// TIA Portal V17 export
// export: Created 2025-05-08T13:17:41.9955383Z, ExportSetting WithDefaults, DisplayName Totally Integrated Automation Portal, DisplayVersion V17 Update 8, DisplayName TIA Portal Openness, DisplayVersion V17 Update 8, DisplayName TIA Portal Version Control Interface, DisplayVersion V17, DisplayName SINAMICS Startdrive Advanced, DisplayVersion V17 SP2, DisplayName SINAMICS Startdrive G110M, G120, G120C, G120D, G120P, G115D, DisplayVersion V17 SP2, DisplayName SINAMICS Startdrive G130, G150, S120, S150, SINAMICS MV, S210, DisplayVersion V17 SP2, DisplayName STEP 7 Professional, DisplayVersion V17 Update 8, DisplayName SINUMERIK ONE STEP 7 Toolbox, DisplayVersion V17 Update 12, DisplayName SINUMERIK 840D sl STEP 7 Toolbox, DisplayVersion V17 Update 12, DisplayName STEP 7 Safety, DisplayVersion V17 Update 6, DisplayName WinCC Advanced, DisplayVersion V17 Update 8
FUNCTION "FC2001_AUTO_SINGLE_SEMI_MANUAL" : Void   // FC2001, LAD
{ S7_Optimized_Access := 'FALSE' }
AUTHOR : ETXETAR
VERSION : 1.0
// stored: AutoNumber false, IsIECCheckEnabled false, SetENOAutomatically false, UDAEnableTagReadback false
   VAR_TEMP
      O_BYTE_0 : Struct   // OPTIONS BYTE 0
         CHANGE_MODE_SEOC_ALARM : Bool;   // CHANGE MODE SEOC ALARM OPTION
         MODE_SELECTED_MEMORY : Bool;   // MODE SELECTED MEMORY OPTION
      END_STRUCT;
      MG1_INPUTS : Struct
         MANUAL : Bool;   // MANUAL INPUT
         SEMIAUTO : Bool;   // SEMIAUTO INPUT
         AUTOMATIC : Bool;   // AUTOMATIC INPUT
         SINGLE : Bool;   // SINGLE INPUT
         NO_MODE : Bool;   // NO MODE INPUT
         JOG : Bool;   // JOG INPUT
         "TOOL CHANGE" : Bool;   // TOOL CHANGE INPUT
      END_STRUCT;
      MG2_INPUTS : Struct
         MANUAL : Bool;   // MANUAL INPUT
         SEMIAUTO : Bool;   // SEMIAUTO INPUT
         AUTOMATIC : Bool;   // AUTOMATIC INPUT
         SINGLE : Bool;   // SINGLE INPUT
         NO_MODE : Bool;   // NO MODE INPUT
         JOG : Bool;   // JOG INPUT
         "TOOL CHANGE" : Bool;   // TOOL CHANGE INPUT
      END_STRUCT;
   END_VAR
   VAR CONSTANT
      FC_NUMBER : Int := 2001;   // NUMBER
   END_VAR
BEGIN

REGION Network 1: OPTIONS OFF
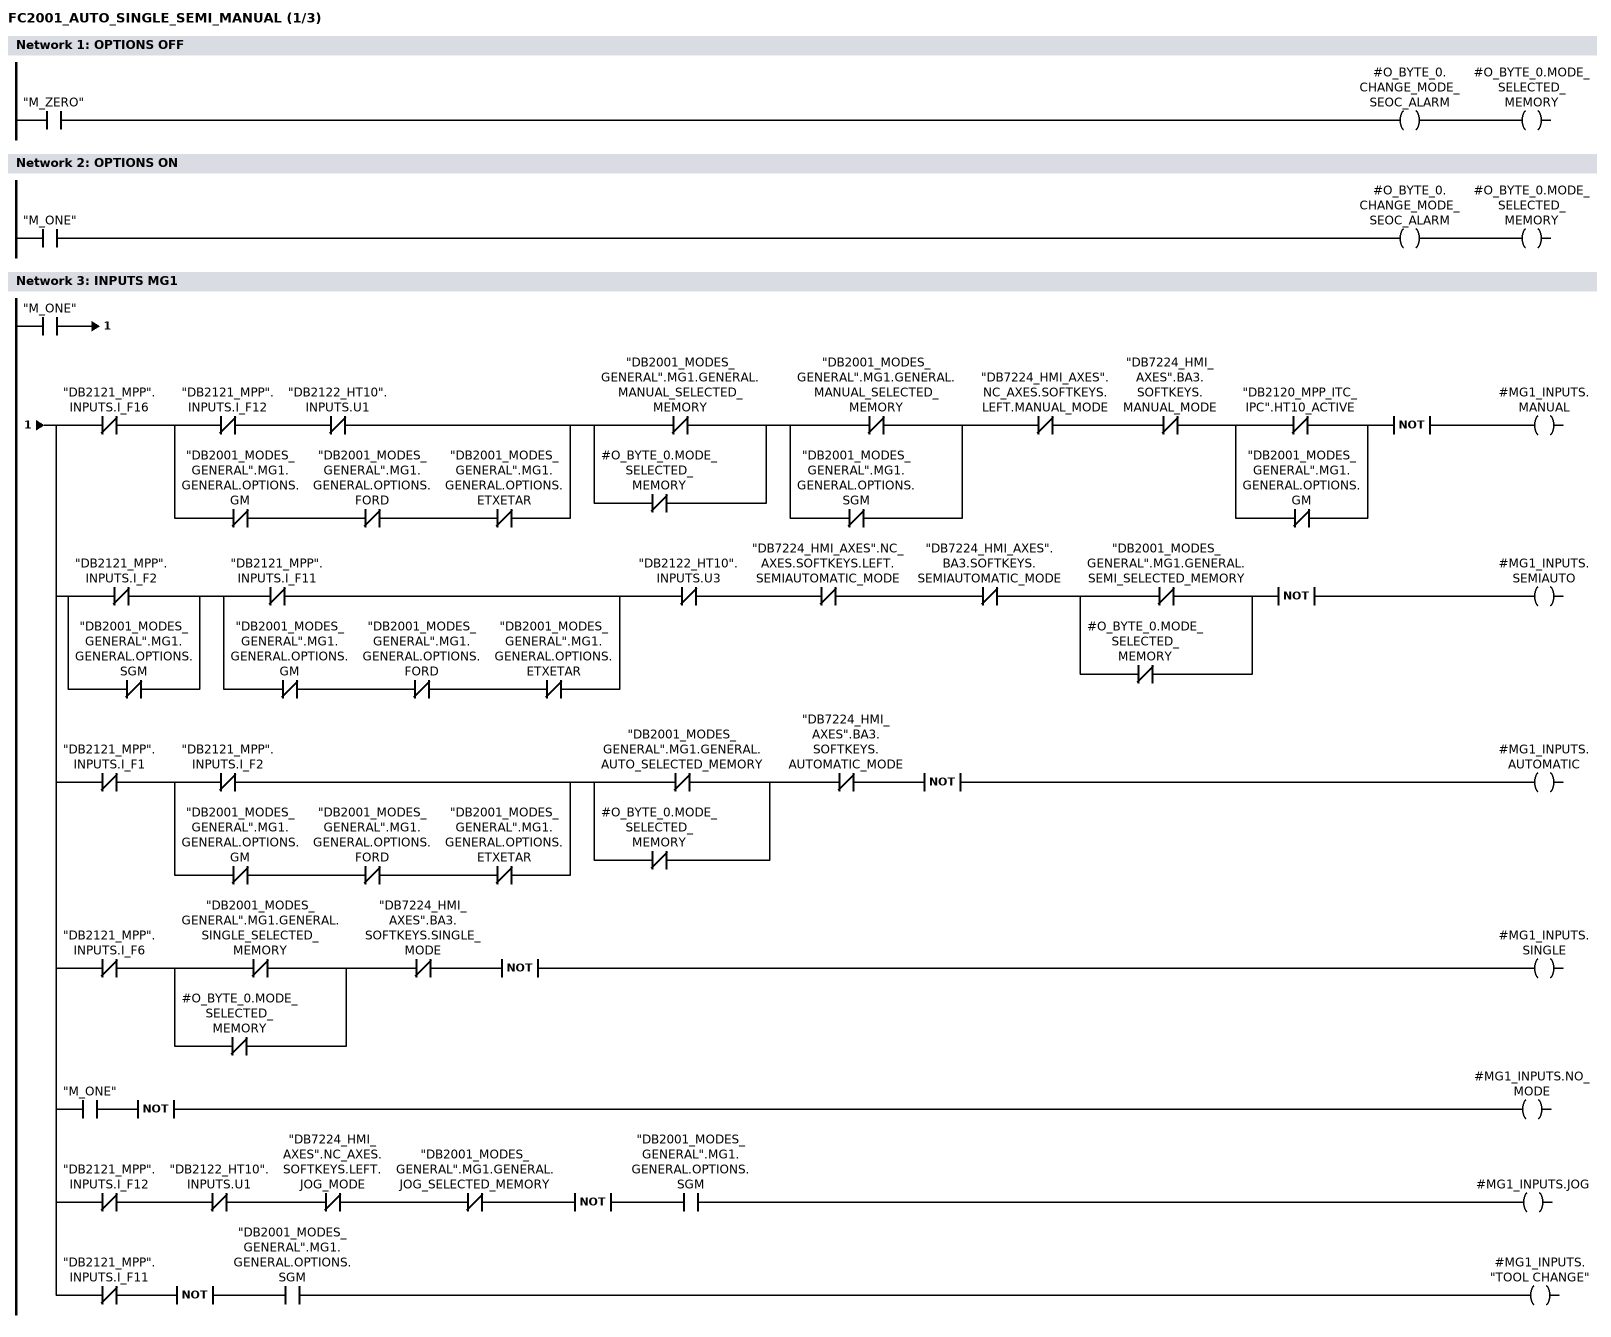
   RUNG wire#powerrail
      Contact( "M_ZERO" )
      Coil( #O_BYTE_0.CHANGE_MODE_SEOC_ALARM )
      Coil( #O_BYTE_0.MODE_SELECTED_MEMORY )
   END_RUNG
   // the same network as SCL:
   #O_BYTE_0.CHANGE_MODE_SEOC_ALARM := "M_ZERO";
   #O_BYTE_0.MODE_SELECTED_MEMORY := "M_ZERO";
END_REGION

REGION Network 2: OPTIONS ON
   RUNG wire#powerrail
      Contact( "M_ONE" )
      Coil( #O_BYTE_0.CHANGE_MODE_SEOC_ALARM )
      Coil( #O_BYTE_0.MODE_SELECTED_MEMORY )
   END_RUNG
   // the same network as SCL:
   #O_BYTE_0.CHANGE_MODE_SEOC_ALARM := "M_ONE";
   #O_BYTE_0.MODE_SELECTED_MEMORY := "M_ONE";
END_REGION

REGION Network 3: INPUTS MG1
   RUNG wire#powerrail
      Contact( "M_ONE" )
      wire#w1
      I_Contact( "DB2121_MPP".INPUTS.I_F16 )
      wire#w2
      I_Contact( "DB2121_MPP".INPUTS.I_F12 )
      I_Contact( "DB2122_HT10".INPUTS.U1 )
      wire#w3
      I_Contact( "DB2001_MODES_GENERAL".MG1.GENERAL.MANUAL_SELECTED_MEMORY )
      wire#w4
      I_Contact( "DB2001_MODES_GENERAL".MG1.GENERAL.MANUAL_SELECTED_MEMORY )
      wire#w5
      I_Contact( "DB7224_HMI_AXES".NC_AXES.SOFTKEYS.LEFT.MANUAL_MODE )
      I_Contact( "DB7224_HMI_AXES".BA3.SOFTKEYS.MANUAL_MODE )
      wire#w6
      I_Contact( "DB2120_MPP_ITC_IPC".HT10_ACTIVE )
      wire#w7
      Not()
      Coil( #MG1_INPUTS.MANUAL )
   END_RUNG
   RUNG wire#w2
      I_Contact( "DB2001_MODES_GENERAL".MG1.GENERAL.OPTIONS.GM )
      I_Contact( "DB2001_MODES_GENERAL".MG1.GENERAL.OPTIONS.FORD )
      I_Contact( "DB2001_MODES_GENERAL".MG1.GENERAL.OPTIONS.ETXETAR )
   END_RUNG wire#w3
   RUNG wire#w3
      I_Contact( #O_BYTE_0.MODE_SELECTED_MEMORY )
   END_RUNG wire#w4
   RUNG wire#w4
      I_Contact( "DB2001_MODES_GENERAL".MG1.GENERAL.OPTIONS.SGM )
   END_RUNG wire#w5
   RUNG wire#w6
      I_Contact( "DB2001_MODES_GENERAL".MG1.GENERAL.OPTIONS.GM )
   END_RUNG wire#w7
   RUNG wire#w1
      I_Contact( "DB2121_MPP".INPUTS.I_F2 )
      wire#w8
      I_Contact( "DB2121_MPP".INPUTS.I_F11 )
      wire#w9
      I_Contact( "DB2122_HT10".INPUTS.U3 )
      I_Contact( "DB7224_HMI_AXES".NC_AXES.SOFTKEYS.LEFT.SEMIAUTOMATIC_MODE )
      I_Contact( "DB7224_HMI_AXES".BA3.SOFTKEYS.SEMIAUTOMATIC_MODE )
      wire#w10
      I_Contact( "DB2001_MODES_GENERAL".MG1.GENERAL.SEMI_SELECTED_MEMORY )
      wire#w11
      Not()
      Coil( #MG1_INPUTS.SEMIAUTO )
   END_RUNG
   RUNG wire#w1
      I_Contact( "DB2001_MODES_GENERAL".MG1.GENERAL.OPTIONS.SGM )
   END_RUNG wire#w8
   RUNG wire#w8
      I_Contact( "DB2001_MODES_GENERAL".MG1.GENERAL.OPTIONS.GM )
      I_Contact( "DB2001_MODES_GENERAL".MG1.GENERAL.OPTIONS.FORD )
      I_Contact( "DB2001_MODES_GENERAL".MG1.GENERAL.OPTIONS.ETXETAR )
   END_RUNG wire#w9
   RUNG wire#w10
      I_Contact( #O_BYTE_0.MODE_SELECTED_MEMORY )
   END_RUNG wire#w11
   RUNG wire#w1
      I_Contact( "DB2121_MPP".INPUTS.I_F1 )
      wire#w12
      I_Contact( "DB2121_MPP".INPUTS.I_F2 )
      wire#w13
      I_Contact( "DB2001_MODES_GENERAL".MG1.GENERAL.AUTO_SELECTED_MEMORY )
      wire#w14
      I_Contact( "DB7224_HMI_AXES".BA3.SOFTKEYS.AUTOMATIC_MODE )
      Not()
      Coil( #MG1_INPUTS.AUTOMATIC )
   END_RUNG
   RUNG wire#w12
      I_Contact( "DB2001_MODES_GENERAL".MG1.GENERAL.OPTIONS.GM )
      I_Contact( "DB2001_MODES_GENERAL".MG1.GENERAL.OPTIONS.FORD )
      I_Contact( "DB2001_MODES_GENERAL".MG1.GENERAL.OPTIONS.ETXETAR )
   END_RUNG wire#w13
   RUNG wire#w13
      I_Contact( #O_BYTE_0.MODE_SELECTED_MEMORY )
   END_RUNG wire#w14
   RUNG wire#w1
      I_Contact( "DB2121_MPP".INPUTS.I_F6 )
      wire#w15
      I_Contact( "DB2001_MODES_GENERAL".MG1.GENERAL.SINGLE_SELECTED_MEMORY )
      wire#w16
      I_Contact( "DB7224_HMI_AXES".BA3.SOFTKEYS.SINGLE_MODE )
      Not()
      Coil( #MG1_INPUTS.SINGLE )
   END_RUNG
   RUNG wire#w15
      I_Contact( #O_BYTE_0.MODE_SELECTED_MEMORY )
   END_RUNG wire#w16
   RUNG wire#w1
      Contact( "M_ONE" )
      Not()
      Coil( #MG1_INPUTS.NO_MODE )
   END_RUNG
   RUNG wire#w1
      I_Contact( "DB2121_MPP".INPUTS.I_F12 )
      I_Contact( "DB2122_HT10".INPUTS.U1 )
      I_Contact( "DB7224_HMI_AXES".NC_AXES.SOFTKEYS.LEFT.JOG_MODE )
      I_Contact( "DB2001_MODES_GENERAL".MG1.GENERAL.JOG_SELECTED_MEMORY )
      Not()
      Contact( "DB2001_MODES_GENERAL".MG1.GENERAL.OPTIONS.SGM )
      Coil( #MG1_INPUTS.JOG )
   END_RUNG
   RUNG wire#w1
      I_Contact( "DB2121_MPP".INPUTS.I_F11 )
      Not()
      Contact( "DB2001_MODES_GENERAL".MG1.GENERAL.OPTIONS.SGM )
      Coil( #MG1_INPUTS."TOOL CHANGE" )
   END_RUNG
   // the same network as SCL:
   #MG1_INPUTS.MANUAL := NOT ("M_ONE" AND NOT "DB2121_MPP".INPUTS.I_F16 AND ((NOT "DB2121_MPP".INPUTS.I_F12 AND NOT "DB2122_HT10".INPUTS.U1) OR (NOT "DB2001_MODES_GENERAL".MG1.GENERAL.OPTIONS.GM AND NOT "DB2001_MODES_GENERAL".MG1.GENERAL.OPTIONS.FORD AND NOT "DB2001_MODES_GENERAL".MG1.GENERAL.OPTIONS.ETXETAR)) AND (NOT "DB2001_MODES_GENERAL".MG1.GENERAL.MANUAL_SELECTED_MEMORY OR NOT #O_BYTE_0.MODE_SELECTED_MEMORY) AND (NOT "DB2001_MODES_GENERAL".MG1.GENERAL.MANUAL_SELECTED_MEMORY OR NOT "DB2001_MODES_GENERAL".MG1.GENERAL.OPTIONS.SGM) AND NOT "DB7224_HMI_AXES".NC_AXES.SOFTKEYS.LEFT.MANUAL_MODE AND NOT "DB7224_HMI_AXES".BA3.SOFTKEYS.MANUAL_MODE AND (NOT "DB2120_MPP_ITC_IPC".HT10_ACTIVE OR NOT "DB2001_MODES_GENERAL".MG1.GENERAL.OPTIONS.GM));
   #MG1_INPUTS.SEMIAUTO := NOT ("M_ONE" AND (NOT "DB2121_MPP".INPUTS.I_F2 OR NOT "DB2001_MODES_GENERAL".MG1.GENERAL.OPTIONS.SGM) AND (NOT "DB2121_MPP".INPUTS.I_F11 OR (NOT "DB2001_MODES_GENERAL".MG1.GENERAL.OPTIONS.GM AND NOT "DB2001_MODES_GENERAL".MG1.GENERAL.OPTIONS.FORD AND NOT "DB2001_MODES_GENERAL".MG1.GENERAL.OPTIONS.ETXETAR)) AND NOT "DB2122_HT10".INPUTS.U3 AND NOT "DB7224_HMI_AXES".NC_AXES.SOFTKEYS.LEFT.SEMIAUTOMATIC_MODE AND NOT "DB7224_HMI_AXES".BA3.SOFTKEYS.SEMIAUTOMATIC_MODE AND (NOT "DB2001_MODES_GENERAL".MG1.GENERAL.SEMI_SELECTED_MEMORY OR NOT #O_BYTE_0.MODE_SELECTED_MEMORY));
   #MG1_INPUTS.AUTOMATIC := NOT ("M_ONE" AND NOT "DB2121_MPP".INPUTS.I_F1 AND (NOT "DB2121_MPP".INPUTS.I_F2 OR (NOT "DB2001_MODES_GENERAL".MG1.GENERAL.OPTIONS.GM AND NOT "DB2001_MODES_GENERAL".MG1.GENERAL.OPTIONS.FORD AND NOT "DB2001_MODES_GENERAL".MG1.GENERAL.OPTIONS.ETXETAR)) AND (NOT "DB2001_MODES_GENERAL".MG1.GENERAL.AUTO_SELECTED_MEMORY OR NOT #O_BYTE_0.MODE_SELECTED_MEMORY) AND NOT "DB7224_HMI_AXES".BA3.SOFTKEYS.AUTOMATIC_MODE);
   #MG1_INPUTS.SINGLE := NOT ("M_ONE" AND NOT "DB2121_MPP".INPUTS.I_F6 AND (NOT "DB2001_MODES_GENERAL".MG1.GENERAL.SINGLE_SELECTED_MEMORY OR NOT #O_BYTE_0.MODE_SELECTED_MEMORY) AND NOT "DB7224_HMI_AXES".BA3.SOFTKEYS.SINGLE_MODE);
   #MG1_INPUTS.NO_MODE := NOT ("M_ONE" AND "M_ONE");
   #MG1_INPUTS.JOG := NOT ("M_ONE" AND NOT "DB2121_MPP".INPUTS.I_F12 AND NOT "DB2122_HT10".INPUTS.U1 AND NOT "DB7224_HMI_AXES".NC_AXES.SOFTKEYS.LEFT.JOG_MODE AND NOT "DB2001_MODES_GENERAL".MG1.GENERAL.JOG_SELECTED_MEMORY) AND "DB2001_MODES_GENERAL".MG1.GENERAL.OPTIONS.SGM;
   #MG1_INPUTS."TOOL CHANGE" := NOT ("M_ONE" AND NOT "DB2121_MPP".INPUTS.I_F11) AND "DB2001_MODES_GENERAL".MG1.GENERAL.OPTIONS.SGM;
END_REGION

REGION Network 4: CALL FB2001 MG1
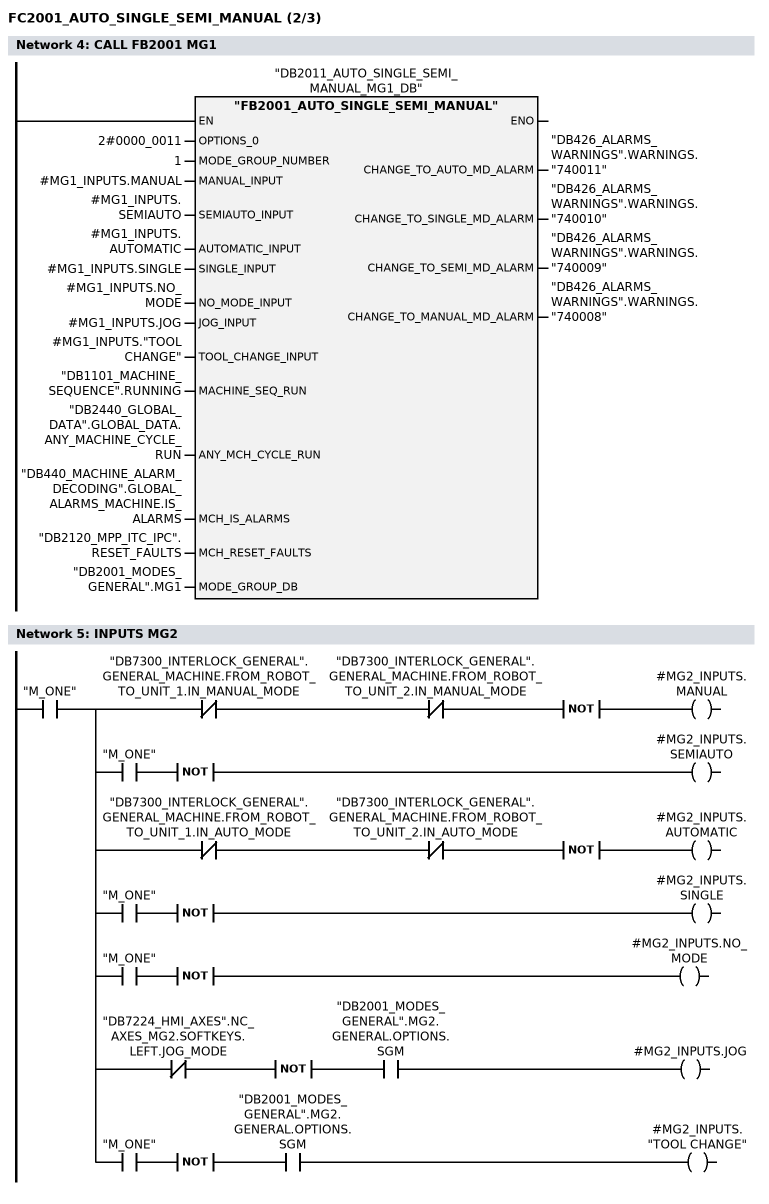
   RUNG wire#powerrail
      "DB2011_AUTO_SINGLE_SEMI_MANUAL_MG1_DB"(OPTIONS_0 := 2#0000_0011, MODE_GROUP_NUMBER := 1, MANUAL_INPUT := #MG1_INPUTS.MANUAL, SEMIAUTO_INPUT := #MG1_INPUTS.SEMIAUTO, AUTOMATIC_INPUT := #MG1_INPUTS.AUTOMATIC, SINGLE_INPUT := #MG1_INPUTS.SINGLE, NO_MODE_INPUT := #MG1_INPUTS.NO_MODE, JOG_INPUT := #MG1_INPUTS.JOG, TOOL_CHANGE_INPUT := #MG1_INPUTS."TOOL CHANGE", MACHINE_SEQ_RUN := "DB1101_MACHINE_SEQUENCE".RUNNING, ANY_MCH_CYCLE_RUN := "DB2440_GLOBAL_DATA".GLOBAL_DATA.ANY_MACHINE_CYCLE_RUN, MCH_IS_ALARMS := "DB440_MACHINE_ALARM_DECODING".GLOBAL_ALARMS_MACHINE.IS_ALARMS, MCH_RESET_FAULTS := "DB2120_MPP_ITC_IPC".RESET_FAULTS, MODE_GROUP_DB := "DB2001_MODES_GENERAL".MG1, CHANGE_TO_AUTO_MD_ALARM => "DB426_ALARMS_WARNINGS".WARNINGS."740011", CHANGE_TO_SINGLE_MD_ALARM => "DB426_ALARMS_WARNINGS".WARNINGS."740010", CHANGE_TO_SEMI_MD_ALARM => "DB426_ALARMS_WARNINGS".WARNINGS."740009", CHANGE_TO_MANUAL_MD_ALARM => "DB426_ALARMS_WARNINGS".WARNINGS."740008")
   END_RUNG
   // the same network as SCL:
   "DB2011_AUTO_SINGLE_SEMI_MANUAL_MG1_DB"(OPTIONS_0 := 2#0000_0011,   // "FB2001_AUTO_SINGLE_SEMI_MANUAL"
                           MODE_GROUP_NUMBER := 1,
                           MANUAL_INPUT := #MG1_INPUTS.MANUAL,
                           SEMIAUTO_INPUT := #MG1_INPUTS.SEMIAUTO,
                           AUTOMATIC_INPUT := #MG1_INPUTS.AUTOMATIC,
                           SINGLE_INPUT := #MG1_INPUTS.SINGLE,
                           NO_MODE_INPUT := #MG1_INPUTS.NO_MODE,
                           JOG_INPUT := #MG1_INPUTS.JOG,
                           TOOL_CHANGE_INPUT := #MG1_INPUTS."TOOL CHANGE",
                           MACHINE_SEQ_RUN := "DB1101_MACHINE_SEQUENCE".RUNNING,
                           ANY_MCH_CYCLE_RUN := "DB2440_GLOBAL_DATA".GLOBAL_DATA.ANY_MACHINE_CYCLE_RUN,
                           MCH_IS_ALARMS := "DB440_MACHINE_ALARM_DECODING".GLOBAL_ALARMS_MACHINE.IS_ALARMS,
                           MCH_RESET_FAULTS := "DB2120_MPP_ITC_IPC".RESET_FAULTS,
                           MODE_GROUP_DB := "DB2001_MODES_GENERAL".MG1,
                           CHANGE_TO_AUTO_MD_ALARM => "DB426_ALARMS_WARNINGS".WARNINGS."740011",
                           CHANGE_TO_SINGLE_MD_ALARM => "DB426_ALARMS_WARNINGS".WARNINGS."740010",
                           CHANGE_TO_SEMI_MD_ALARM => "DB426_ALARMS_WARNINGS".WARNINGS."740009",
                           CHANGE_TO_MANUAL_MD_ALARM => "DB426_ALARMS_WARNINGS".WARNINGS."740008");
END_REGION

REGION Network 5: INPUTS MG2
   RUNG wire#powerrail
      Contact( "M_ONE" )
      wire#w1
      I_Contact( "DB7300_INTERLOCK_GENERAL".GENERAL_MACHINE.FROM_ROBOT_TO_UNIT_1.IN_MANUAL_MODE )
      I_Contact( "DB7300_INTERLOCK_GENERAL".GENERAL_MACHINE.FROM_ROBOT_TO_UNIT_2.IN_MANUAL_MODE )
      Not()
      Coil( #MG2_INPUTS.MANUAL )
   END_RUNG
   RUNG wire#w1
      Contact( "M_ONE" )
      Not()
      Coil( #MG2_INPUTS.SEMIAUTO )
   END_RUNG
   RUNG wire#w1
      I_Contact( "DB7300_INTERLOCK_GENERAL".GENERAL_MACHINE.FROM_ROBOT_TO_UNIT_1.IN_AUTO_MODE )
      I_Contact( "DB7300_INTERLOCK_GENERAL".GENERAL_MACHINE.FROM_ROBOT_TO_UNIT_2.IN_AUTO_MODE )
      Not()
      Coil( #MG2_INPUTS.AUTOMATIC )
   END_RUNG
   RUNG wire#w1
      Contact( "M_ONE" )
      Not()
      Coil( #MG2_INPUTS.SINGLE )
   END_RUNG
   RUNG wire#w1
      Contact( "M_ONE" )
      Not()
      Coil( #MG2_INPUTS.NO_MODE )
   END_RUNG
   RUNG wire#w1
      I_Contact( "DB7224_HMI_AXES".NC_AXES_MG2.SOFTKEYS.LEFT.JOG_MODE )
      Not()
      Contact( "DB2001_MODES_GENERAL".MG2.GENERAL.OPTIONS.SGM )
      Coil( #MG2_INPUTS.JOG )
   END_RUNG
   RUNG wire#w1
      Contact( "M_ONE" )
      Not()
      Contact( "DB2001_MODES_GENERAL".MG2.GENERAL.OPTIONS.SGM )
      Coil( #MG2_INPUTS."TOOL CHANGE" )
   END_RUNG
   // the same network as SCL:
   #MG2_INPUTS.MANUAL := NOT ("M_ONE" AND NOT "DB7300_INTERLOCK_GENERAL".GENERAL_MACHINE.FROM_ROBOT_TO_UNIT_1.IN_MANUAL_MODE AND NOT "DB7300_INTERLOCK_GENERAL".GENERAL_MACHINE.FROM_ROBOT_TO_UNIT_2.IN_MANUAL_MODE);
   #MG2_INPUTS.SEMIAUTO := NOT ("M_ONE" AND "M_ONE");
   #MG2_INPUTS.AUTOMATIC := NOT ("M_ONE" AND NOT "DB7300_INTERLOCK_GENERAL".GENERAL_MACHINE.FROM_ROBOT_TO_UNIT_1.IN_AUTO_MODE AND NOT "DB7300_INTERLOCK_GENERAL".GENERAL_MACHINE.FROM_ROBOT_TO_UNIT_2.IN_AUTO_MODE);
   #MG2_INPUTS.SINGLE := NOT ("M_ONE" AND "M_ONE");
   #MG2_INPUTS.NO_MODE := NOT ("M_ONE" AND "M_ONE");
   #MG2_INPUTS.JOG := NOT ("M_ONE" AND NOT "DB7224_HMI_AXES".NC_AXES_MG2.SOFTKEYS.LEFT.JOG_MODE) AND "DB2001_MODES_GENERAL".MG2.GENERAL.OPTIONS.SGM;
   #MG2_INPUTS."TOOL CHANGE" := NOT ("M_ONE" AND "M_ONE") AND "DB2001_MODES_GENERAL".MG2.GENERAL.OPTIONS.SGM;
END_REGION

REGION Network 6: CALL FB2001 MG1
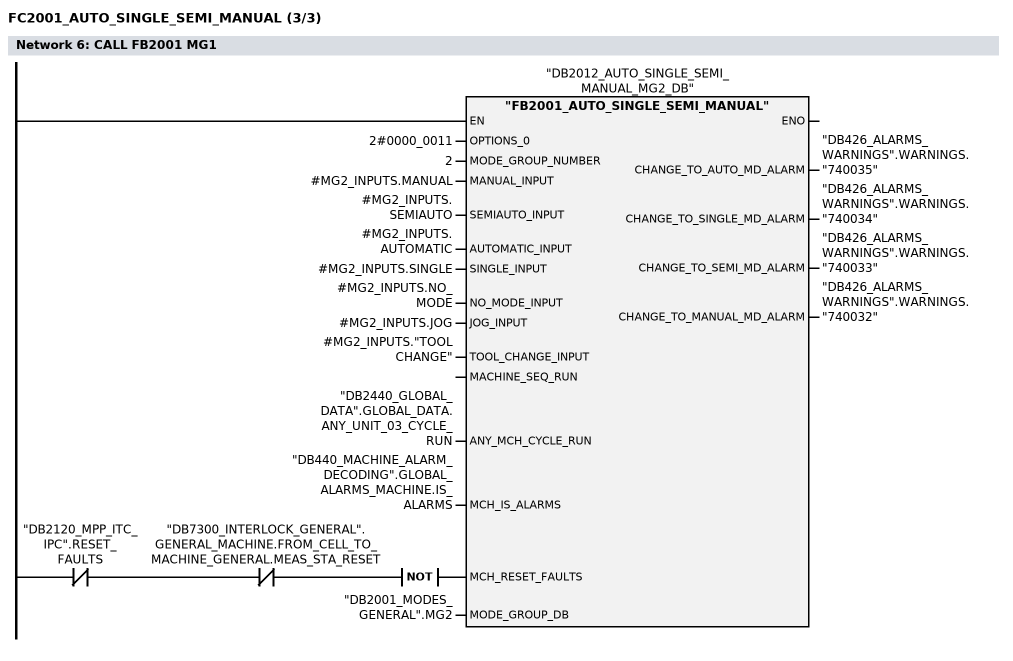
   RUNG wire#powerrail
      "DB2012_AUTO_SINGLE_SEMI_MANUAL_MG2_DB"(MCH_RESET_FAULTS := wire#w1, OPTIONS_0 := 2#0000_0011, MODE_GROUP_NUMBER := 2, MANUAL_INPUT := #MG2_INPUTS.MANUAL, SEMIAUTO_INPUT := #MG2_INPUTS.SEMIAUTO, AUTOMATIC_INPUT := #MG2_INPUTS.AUTOMATIC, SINGLE_INPUT := #MG2_INPUTS.SINGLE, NO_MODE_INPUT := #MG2_INPUTS.NO_MODE, JOG_INPUT := #MG2_INPUTS.JOG, TOOL_CHANGE_INPUT := #MG2_INPUTS."TOOL CHANGE", MACHINE_SEQ_RUN :=, ANY_MCH_CYCLE_RUN := "DB2440_GLOBAL_DATA".GLOBAL_DATA.ANY_UNIT_03_CYCLE_RUN, MCH_IS_ALARMS := "DB440_MACHINE_ALARM_DECODING".GLOBAL_ALARMS_MACHINE.IS_ALARMS, MODE_GROUP_DB := "DB2001_MODES_GENERAL".MG2, CHANGE_TO_AUTO_MD_ALARM => "DB426_ALARMS_WARNINGS".WARNINGS."740035", CHANGE_TO_SINGLE_MD_ALARM => "DB426_ALARMS_WARNINGS".WARNINGS."740034", CHANGE_TO_SEMI_MD_ALARM => "DB426_ALARMS_WARNINGS".WARNINGS."740033", CHANGE_TO_MANUAL_MD_ALARM => "DB426_ALARMS_WARNINGS".WARNINGS."740032")
   END_RUNG
   RUNG wire#powerrail
      I_Contact( "DB2120_MPP_ITC_IPC".RESET_FAULTS )
      I_Contact( "DB7300_INTERLOCK_GENERAL".GENERAL_MACHINE.FROM_CELL_TO_MACHINE_GENERAL.MEAS_STA_RESET )
      Not()
   END_RUNG wire#w1
   // the same network as SCL:
   "DB2012_AUTO_SINGLE_SEMI_MANUAL_MG2_DB"(OPTIONS_0 := 2#0000_0011,   // "FB2001_AUTO_SINGLE_SEMI_MANUAL"
                           MODE_GROUP_NUMBER := 2,
                           MANUAL_INPUT := #MG2_INPUTS.MANUAL,
                           SEMIAUTO_INPUT := #MG2_INPUTS.SEMIAUTO,
                           AUTOMATIC_INPUT := #MG2_INPUTS.AUTOMATIC,
                           SINGLE_INPUT := #MG2_INPUTS.SINGLE,
                           NO_MODE_INPUT := #MG2_INPUTS.NO_MODE,
                           JOG_INPUT := #MG2_INPUTS.JOG,
                           TOOL_CHANGE_INPUT := #MG2_INPUTS."TOOL CHANGE",
                           ANY_MCH_CYCLE_RUN := "DB2440_GLOBAL_DATA".GLOBAL_DATA.ANY_UNIT_03_CYCLE_RUN,
                           MCH_IS_ALARMS := "DB440_MACHINE_ALARM_DECODING".GLOBAL_ALARMS_MACHINE.IS_ALARMS,
                           MCH_RESET_FAULTS := NOT (NOT "DB2120_MPP_ITC_IPC".RESET_FAULTS AND NOT "DB7300_INTERLOCK_GENERAL".GENERAL_MACHINE.FROM_CELL_TO_MACHINE_GENERAL.MEAS_STA_RESET),
                           MODE_GROUP_DB := "DB2001_MODES_GENERAL".MG2,
                           CHANGE_TO_AUTO_MD_ALARM => "DB426_ALARMS_WARNINGS".WARNINGS."740035",
                           CHANGE_TO_SINGLE_MD_ALARM => "DB426_ALARMS_WARNINGS".WARNINGS."740034",
                           CHANGE_TO_SEMI_MD_ALARM => "DB426_ALARMS_WARNINGS".WARNINGS."740033",
                           CHANGE_TO_MANUAL_MD_ALARM => "DB426_ALARMS_WARNINGS".WARNINGS."740032");
END_REGION
END_FUNCTION
